FUNCTION_BLOCK horimetro2 (* Composite Function Block Type - Horimetro com persistencia funcional *)
  (* Standard: 61499-2 *)
  (* Version 1.0.0, 11/05/2026, Hidryco, Hidryco, Versao corrigida do horimetro - PERSISTENCE.outputN agora alimenta basicHorimetro2.INIT_xxx para restaurar contagem apos reinicio do PLC *)
  PACKAGE Hidryco.HidrycoLib;
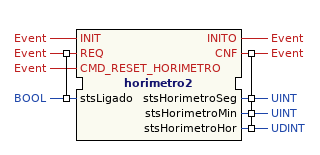
  EVENT_INPUT
    INIT; (* Inicializacao *)
    REQ WITH stsLigado; (* Pulso de 1s *)
    CMD_RESET_HORIMETRO; (* Zera o horimetro *)
  END_EVENT
  EVENT_OUTPUT
    INITO; (* Confirmacao de inicializacao *)
    CNF WITH stsHorimetroSeg, stsHorimetroMin, stsHorimetroHor; (* Confirmacao de execucao *)
  END_EVENT
  VAR_INPUT
    stsLigado : BOOL; (* 1 = equipamento ligado (acumula tempo) *)
  END_VAR
  VAR_OUTPUT
    stsHorimetroSeg : UINT; (* Segundos (0..59) *)
    stsHorimetroMin : UINT; (* Minutos (0..59) *)
    stsHorimetroHor : UDINT; (* Horas totais *)
  END_VAR
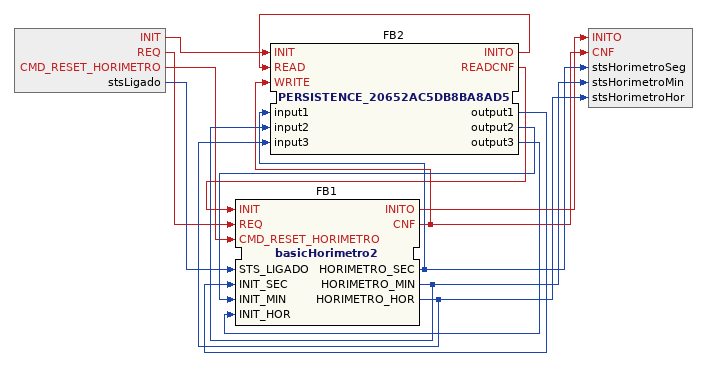
  FBS
    FB1 : basicHorimetro2;
    FB2 : PERSISTENCE_20652AC5DB8BA8AD5; {SET_ATTRIBUTE(Configuration.GenericFBType.InterfaceParams, Runtime.Standard#I:=3;input${I$}:UINT,UINT,UDINT)}
  END_FBS
  EVENT_CONNECTIONS
    INIT TO FB2.INIT;
    FB2.INITO TO FB2.READ;
    FB2.READCNF TO FB1.INIT;
    FB1.INITO TO INITO;
    REQ TO FB1.REQ;
    CMD_RESET_HORIMETRO TO FB1.CMD_RESET_HORIMETRO;
    FB1.CNF TO FB2.WRITE;
    FB1.CNF TO CNF;
  END_CONNECTIONS
  DATA_CONNECTIONS
    stsLigado TO FB1.STS_LIGADO;
    FB2.output1 TO FB1.INIT_SEC;
    FB2.output2 TO FB1.INIT_MIN;
    FB2.output3 TO FB1.INIT_HOR;
    FB1.HORIMETRO_SEC TO stsHorimetroSeg;
    FB1.HORIMETRO_MIN TO stsHorimetroMin;
    FB1.HORIMETRO_HOR TO stsHorimetroHor;
    FB1.HORIMETRO_SEC TO FB2.input1;
    FB1.HORIMETRO_MIN TO FB2.input2;
    FB1.HORIMETRO_HOR TO FB2.input3;
  END_CONNECTIONS
END_FUNCTION_BLOCK
